VISUALIZATION Controlbox  // 2x2
END_VISUALIZATION

(* stored: Version 1.1.0.1, ProductVersion 3.1.4024.12
   Visu Controlbox: Id {37c99271-e1ca-49d5-935b-2ab9689d1605} *)
